FUNCTION TryConvert_BYTE_TO_LWORD : BOOL
VAR_INPUT
	in : BYTE;
	out : REFERENCE TO LWORD;
END_VAR

out := BYTE_TO_LWORD(in);
TryConvert_BYTE_TO_LWORD := TRUE;

END_FUNCTION

(* stored: Version 1.1.0.1, ProductVersion 3.1.4024.12
   POU TryConvert_BYTE_TO_LWORD: Id {1a4d5ea9-bacd-40d0-aaf5-a1f1abe5d617}, SpecialFunc None *)
